// TIA Portal V20 export
DATA_BLOCK "LPFE_DigitalEventConfig"   // DB251
TITLE = LPFE_DigitalEventConfig
AUTHOR : DI FA SUP
FAMILY : LPFE
// Contains the digital event handler configuration and Rootcause alarm information
// stored: Access Published, MemoryReserve 100, Namespace PFE
   VAR
      AlarmsDisplayClass : Array[0..31] of UInt;   // Display classes that are going to be processed by Get Alarm Block
      RootcauseCellData : Array[0.._.NO_OF_CELLS] of "LPFE_typeRootCauseCellData";   // Rootcause data stored when the rootacause filter is enabled in the digital event
   END_VAR
BEGIN
   AlarmsDisplayClass[0] := 0;
   AlarmsDisplayClass[1] := 1;
   AlarmsDisplayClass[2] := 2;
   AlarmsDisplayClass[3] := 3;
   AlarmsDisplayClass[4] := 4;
   AlarmsDisplayClass[5] := 5;
   AlarmsDisplayClass[6] := 6;
   AlarmsDisplayClass[7] := 7;
   AlarmsDisplayClass[8] := 8;
   AlarmsDisplayClass[9] := 9;
   AlarmsDisplayClass[10] := 10;
   AlarmsDisplayClass[11] := 11;
   AlarmsDisplayClass[12] := 12;
   AlarmsDisplayClass[13] := 13;
   AlarmsDisplayClass[14] := 14;
   AlarmsDisplayClass[15] := 15;
   AlarmsDisplayClass[16] := 16;
   AlarmsDisplayClass[17..31] := 256;
END_DATA_BLOCK
